FUNCTION_BLOCK FB_DriveSimpleDoor IMPLEMENTS IF_DriveConstVel
VAR_INPUT
	bLimitSwitchOpen, bLimitSwitchClosed : BOOL;		(* Limit switches fpr door open and door closed *)
END_VAR
VAR_OUTPUT
	bDriveEnable, bOpen, bClose : BOOL;					(* Door drive enable, input signals for operning and closing the door *)
END_VAR
VAR
END_VAR

METHOD doorClose : BOOL
(* Close door *)
bClose := TRUE;						(* set outputs for door drive, requires bDoorEnable = TRUE *)
bOpen := FALSE;

doorClose := bLimitSwitchClosed;	(* TRUE if and only if limit switch is TRUE *)
END_METHOD

METHOD doorDisable
bDriveEnable := FALSE;
END_METHOD

METHOD doorEnable
bDriveEnable := TRUE;
END_METHOD

METHOD doorOpen : BOOL
(* Open door *)
bOpen := TRUE;					(* set outputs for door drive, requires bDoorEnable = TRUE *)
bClose := FALSE;

doorOpen := bLimitSwitchOpen;	(* TRUE if and only if limit switch is TRUE *)
END_METHOD

END_FUNCTION_BLOCK

(* stored: Version 1.1.0.1, ProductVersion 3.1.4024.6
   POU FB_DriveSimpleDoor: Id {6c6f7b46-3a89-4f17-95b1-055e80ffbab5}, SpecialFunc None
   Method doorClose: Id {58f9614e-cc91-4a6f-aaa6-0428fd8245e1}
   Method doorDisable: Id {6d0113df-a5ad-449c-8dbc-48fdf8233374}
   Method doorEnable: Id {0ae92346-b43f-480f-8e96-8197df7689c8}
   Method doorOpen: Id {946036e9-b71e-4e43-9072-1dd3d6f022b1} *)
